{attribute 'qualified_only'}
VAR_GLOBAL
END_VAR

(* stored: Version 1.1.0.1, ProductVersion 3.1.4026.17
   GVL GVL_BALLAST: Id {0676789c-ef16-4b1f-a59c-8284102d598d} *)
